(* IEC 61131-3 sources: mp-conveyorbelt/test/Process, 2 files *)

(* ---- test.st ---- *)
NAMESPACE Simatic.Ax.xxx
    USING AxUnit.Assert;

    NAMESPACE Simatic.Ax.Test

        {TestFixture}
        CLASS test22

            {Test}
            METHOD PUBLIC MyMethod
                 // write your test code here
                 Equal(expected := TRUE, actual := TRUE);
                ;
            END_METHOD
        END_CLASS
    END_NAMESPACE
END_NAMESPACE

(* ---- TestProcess.st ---- *)
USING Simatic.Ax.IO.Input;
USING Simatic.Ax.Dynamics;

NAMESPACE Simatic.Ax.Process

    {TestFixture}
    CLASS MyTestFixture
        VAR PRIVATE
            timeProvider : ConstantTimeProvider := (seconds := 0.02);
            p : ProcessHandler;
            pStateLess : ProcessHandler;
            risingSignalMock : BinSignalRisingEdgeMock;
            fallingSignalMock : BinSignalFallingEdgeMock;
        END_VAR

        {TestSetup}
        METHOD PUBLIC TestSetup
            p := pStateLess;
            p.TimeProvider := timeProvider;
        END_METHOD

        {Test} // This test checks the finished process on falling edge of the next clock signal
        METHOD PUBLIC Process_Finished_OnfallingEdgeOfMachineClock  // change to falling edge
            p.machineClock := fallingSignalMock;
            p.Start();
            AxUnit.Assert.Equal(actual := p.GetState(), expected := ProcessState#Fill);
            p.Execute();
            AxUnit.Assert.Equal(actual := p.GetState(), expected := ProcessState#Unfill);
        END_METHOD
    END_CLASS

    /// Mock the rising edge of the signal
    CLASS BinSignalRisingEdgeMock
        IMPLEMENTS ItfBinSignal
        VAR
        END_VAR

        METHOD PUBLIC Q : BOOL
            Q := TRUE;
        END_METHOD

        METHOD PUBLIC QRis : BOOL
            QRis := TRUE;
        END_METHOD

        METHOD PUBLIC QFal : BOOL
            QFal := FALSE;
        END_METHOD

        METHOD PUBLIC QBad : BOOL
            QBad := FALSE;
        END_METHOD
    END_CLASS

    /// Mock the falling edge of the signal
    CLASS BinSignalFallingEdgeMock
        IMPLEMENTS ItfBinSignal
        VAR
        END_VAR

        METHOD PUBLIC Q : BOOL
            Q := FALSE;
        END_METHOD

        METHOD PUBLIC QRis : BOOL
            QRis := FALSE;
        END_METHOD

        METHOD PUBLIC QFal : BOOL
            QFal := TRUE;
        END_METHOD

        METHOD PUBLIC QBad : BOOL
            QBad := FALSE;
        END_METHOD
    END_CLASS

END_NAMESPACE
